{library PUBLIC}
(* Level 1 function to get communication status for a specific address.

   Depending on the address (specific device) different status checks can be performed, e.g., bus status.
   Note that this function does not transmit any data to check the real status of a device it only check if it is possible to communicate.
   On success true is returned otherwise false.
*)
FUNCTION NodeGetStatus : BOOL
VAR_INPUT
	Address: 		INT;		(* Address, use the function ToAddress() to convert station and device number to a valid address. *)
END_VAR
VAR
END_VAR

NodeGetStatus:=FALSE;

IF _CheckInstance(Address) THEN
	NodeGetStatus:=TRUE;

	(* Code here to check bus status *)
END_IF;

END_FUNCTION

(* stored: Version 1.1.0.1, ProductVersion 3.1.4024.2
   POU NodeGetStatus: Id {d5d32d84-365a-4395-9730-2f3155d93460}, SpecialFunc None *)
